FUNCTION_BLOCK Mc3MotionCoupleTask_Gearing EXTENDS Mc3MotionTask
VAR
	McGearIn				  : Tc3_Mc3Ptp.MC_GearIn;
	_InGear					  : BOOL;
	_RatioNumerator			  : LREAL := 1.0;
	_RatioDenominator		  : LREAL := 1.0;
	DummyAxis				  : Tc3_Mc3Ptp.AXIS_REF;
	MasterAxis				  : REFERENCE TO Tc3_Mc3Ptp.AXIS_REF;
	_Master					  : I_Mc3Axis;
	_McBufferMode			  : Tc3_Mc3Ptp.EBufferMode;
END_VAR

PROPERTY BufferMode : Tc3_Mc3Ptp.EBufferMode
SET
_McBufferMode := BufferMode;
END_SET
END_PROPERTY

{attribute 'monitoring' := 'call'}
PROPERTY Busy : BOOL
GET
Busy := McGearIn.Busy;
END_GET
END_PROPERTY

METHOD CyclicLogic
McGearIn(Master			:= MasterAxis,
		 Slave			:= _Axis.Axis,
		 Acceleration	:= _Axis.Acceleration,
		 Deceleration	:= _Axis.Deceleration,
		 Jerk			:= _Axis.Jerk,
		 BufferMode		:= _McBufferMode,
		 InGear			=> _InGear,
		 Busy			=>,
		 Active			=>,
		 CommandAborted =>,
		 Error			=>,
		 ErrorId		=>,
		 MasterHasError =>);

McGearIn.Execute := FALSE;
END_METHOD

{attribute 'monitoring' := 'call'}
PROPERTY Error : BOOL
GET
Error := McGearIn.Error;
END_GET
END_PROPERTY

{attribute 'monitoring' := 'call'}
PROPERTY ErrorId : UDINT
GET
ErrorId := McGearIn.ErrorID;
END_GET
END_PROPERTY

METHOD Execute : BOOL
IF NOT McGearIn.Active THEN
	IF _Axis.Error OR Busy THEN
		RETURN;
	END_IF

	McGearIn(Master			:= MasterAxis,
			 Execute		:= TRUE,
			 Slave			:= _Axis.Axis,
			 Acceleration	:= _Axis.Acceleration,
			 Deceleration	:= _Axis.Deceleration,
			 Jerk			:= _Axis.Jerk,
			 BufferMode		:= _McBufferMode,
			 InGear			=> _InGear,
			 Busy			=>,
			 Active			=>,
			 CommandAborted =>,
			 Error			=>,
			 ErrorId		=>,
			 MasterHasError =>);
END_IF

Execute := TRUE;
END_METHOD

{attribute 'monitoring' := 'call'}
PROPERTY InGear : BOOL
GET
InGear := _InGear;
END_GET
END_PROPERTY

PROPERTY Master : I_Mc3Axis
SET
_Master := Master;
IF _Master <> 0 THEN
	MasterAxis REF= _Master.Axis;
ELSE
	MasterAxis REF= DummyAxis;
END_IF
END_SET
END_PROPERTY

{attribute 'monitoring' := 'call'}
PROPERTY MasterHasError : BOOL
GET
MasterHasError := McGearIn.MasterHasError;
END_GET
END_PROPERTY

{attribute 'monitoring' := 'call'}
PROPERTY RatioDenominator : LREAL
SET
_RatioDenominator := RatioDenominator;
END_SET
END_PROPERTY

{attribute 'monitoring' := 'call'}
PROPERTY RatioNumerator : LREAL
SET
_RatioNumerator := RatioNumerator;
END_SET
END_PROPERTY

PROPERTY ReactionToMasterError : EReactionToMasterError
SET
McGearIn.ReactionToMasterError := ReactionToMasterError;
END_SET
END_PROPERTY

PROPERTY ReactionToSlaveError : EReactionToSlaveError
SET
McGearIn.ReactionToSlaveError := ReactionToSlaveError;
END_SET
END_PROPERTY

END_FUNCTION_BLOCK

(* stored: Version 1.1.0.1, ProductVersion 3.1.4026.20
   POU Mc3MotionCoupleTask_Gearing: Id {2f4484a1-c944-4a29-90ac-f5924635f2f1}, SpecialFunc None
   Property BufferMode: Id {fc1ef0f7-3adf-4392-8119-101122a63baf}
   Set Set: Id {c1b84a64-70f6-438d-a446-e4c0d65bff1b}
   Property Busy: Id {f0016e11-0a74-43bb-a633-efb15fa73cf6}
   Get Get: Id {0e4c5633-d901-4fac-a304-b0ec3843442e}
   Method CyclicLogic: Id {337e3a01-93fb-4c7e-a97e-13d009ee1a39}
   Property Error: Id {c40afe1b-b7d4-42f8-8ee8-94335d915a03}
   Get Get: Id {379b9653-db4f-4788-9bd4-12200b00c6f5}
   Property ErrorId: Id {4041ce7a-adf8-4ec3-99f0-ac2439b34c6f}
   Get Get: Id {f8c988ab-a175-46a9-9eb4-4e5bc221e9e7}
   Method Execute: Id {ed28c839-8f67-40eb-aaad-6b389c70ca56}
   Property InGear: Id {63aeaec5-6f7f-4ff2-8190-086b9f67ad44}
   Get Get: Id {93bdd8ba-23d4-4a46-99f3-f1db44ae0af9}
   Property Master: Id {193f744e-04f2-4f86-ae67-cc9a2de68cc3}
   Set Set: Id {51cd390a-4966-47b3-bd0a-66643001bc22}
   Property MasterHasError: Id {73723358-b24a-447f-9873-159a29114431}
   Get Get: Id {858eb977-eaf1-41ac-8534-206c5e022461}
   Property RatioDenominator: Id {12c9ae14-9d32-434c-a275-1b3e82dbeafb}
   Set Set: Id {99467d9a-fbd5-4581-897d-65ef07609208}
   Property RatioNumerator: Id {348ae990-2cef-4379-aa55-ad15c8a94ccf}
   Set Set: Id {51db2914-c08e-49f1-adff-1504aed61cf3}
   Property ReactionToMasterError: Id {d19df0f0-5909-491e-b473-7a9fa5f5aeb7}
   Set Set: Id {5bfc2ff6-df72-4738-b4b8-4113eb5fef0e}
   Property ReactionToSlaveError: Id {af31d6c3-a8ca-435c-977f-9db4eb3cf1c9}
   Set Set: Id {cc5a8f87-25fe-4f63-a8cf-61ac2b9f82a3} *)
